(* IEC 61131-3 sources: Lasal/CPU_5344_V01/Class/punchToolSettingsMpsControl, 1 file *)

(* ---- punchToolSettingsMpsControl.st ---- *)
(*!
<Class
	Name               = "punchToolSettingsMpsControl"
	Revision           = "1.0"
	RealtimeTask       = "false"
	CyclicTask         = "false"
	BackgroundTask     = "false"
	Sigmatek           = "false"
	OSInterface        = "false"
	HighPriority       = "false"
	Automatic          = "false"
	UpdateMode         = "Prescan"
	SharedCommandTable = "true"
	Objectsize         = "(284,120)">
	<Channels>
		<Server Name="setting1" Visualized="true" Initialize="false" WriteProtected="true" Retentive="false"/>
		<Client Name="offset" Required="true" Internal="false"/>
	</Channels>
	<Network Name="punchToolSettingsMpsControl">
		<!-- List of Components in this network -->
		<Components>
			<Object
				Name       = "_base"
				Class      = "baseToolSettingsMpsControl"
				Position   = "(218,120)"
				Visualized = "true"
				Remotely   = "true">
				<Channels>
					<Server Name="amountOfSettings" Value="4"/>
					<Server Name="ClassSvr"/>
					<Server Name="Name"/>
					<Server Name="plane" Value="right"/>
					<Server Name="toolType" Value="9"/>
				</Channels>
			</Object>
		</Components>
		<Comments>
		</Comments>
		<!-- List of Connections in this network -->
		<Connections>
			<Connection Source="this.ClassSvr" Destination="_base.ClassSvr" Vertices="(690,210),(518,210),"/>
			<Connection Source="this.toolType" Destination="_base.toolType" Vertices="(690,270),(518,270),"/>
			<Connection Source="this.Name" Destination="_base.Name" Vertices="(690,330),(518,330),"/>
			<Connection Source="this.plane" Destination="_base.plane" Vertices="(690,390),(518,390),"/>
			<Connection Source="this.amountOfSettings" Destination="_base.amountOfSettings" Vertices="(690,450),(518,450),"/>
		</Connections>
		<!-- Headerfiles -->
		<Options>
		</Options>
	</Network>
</Class>
*)
#pragma using baseToolSettingsMpsControl

punchToolSettingsMpsControl : CLASS
: baseToolSettingsMpsControl
  //Servers:
	setting1 	: SvrCh_DINT;
  //Clients:
	offset 	: CltCh_DINT;
  //Variables:
  //Functions:

	FUNCTION VIRTUAL GLOBAL setting1::Read
		VAR_OUTPUT
			output (EAX) 	: DINT;
		END_VAR;
  //Tables:
	FUNCTION @STD
		VAR_OUTPUT
			ret_code	: CONFSTATES;
		END_VAR;
	FUNCTION GLOBAL TAB @CT_;
END_CLASS;

FUNCTION VIRTUAL GLOBAL punchToolSettingsMpsControl::setting1::Read
	VAR_OUTPUT
		output (EAX) 	: DINT;
	END_VAR

  offset:= offset.Read();
  setting1:= offset;

	output := setting1;

END_FUNCTION
